DATA_BLOCK "SafetyInterlock_DB"
{ S7_Optimized_Access := 'FALSE' }
VERSION : 0.1
NON_RETAIN
   VAR
      SystemSafetyInterlock : Bool := TRUE;   // 系统级安全联锁状态
      EmergencyStopActive : Bool;   // 紧急停止激活
      MainPowerFault : Bool;   // 主电源故障
      SafetyDoorOpen : Bool;   // 安全门打开

      DeviceSafetyInterlock : Struct   // 设备安全联锁
         CompressorSafetyInterlock : Bool := TRUE;   // 压缩机安全联锁
         ChillerSafetyInterlock : Bool := TRUE;   // 冷水机安全联锁
         PumpSafetyInterlock : Bool := TRUE;   // 水泵安全联锁
         FanSafetyInterlock : Bool := TRUE;   // 风机安全联锁
      END_STRUCT;

      ValveSafetyInterlock : Struct   // 阀门安全联锁
         MainGasValveSafetyInterlock : Bool := TRUE;   // 主气路阀门安全联锁
         PurgingValveSafetyInterlock : Bool := TRUE;   // 吹扫阀门安全联锁
         CoolingValveSafetyInterlock : Bool := TRUE;   // 冷却阀门安全联锁
      END_STRUCT;



   END_VAR

BEGIN

END_DATA_BLOCK